INTERFACE IReadOnlyAnalogAnalogInput EXTENDS TOF_Automation.IInputLeafAutomationComponent, TOF_Core.IIOBindable

{attribute 'monitoring' := 'call'}
PROPERTY Converter : IAnalogValueConverter
GET
END_GET
END_PROPERTY

{attribute 'monitoring' := 'call'}
PROPERTY RawValue : LREAL
GET
END_GET
END_PROPERTY

{attribute 'monitoring' := 'call'}
PROPERTY FINAL RawValueType : RAW_ANALOG_VALUE_TYPE
GET
END_GET
END_PROPERTY

{attribute 'monitoring' := 'call'}
PROPERTY Status : REFERENCE TO ANALOG_INPUT_STATUS
GET
END_GET
END_PROPERTY

{attribute 'monitoring' := 'call'}
PROPERTY Value : LREAL
GET
END_GET
END_PROPERTY

END_INTERFACE

(* stored: Version 1.1.0.1
   Itf IReadOnlyAnalogAnalogInput: Id {f18291d7-6e1e-47c5-9cfe-5eb8b3628862}
   Property Converter: Id {38183ee6-a347-4153-bc4c-2d175e7d5e33}
   Get Get: Id {c478d920-13fd-4460-a2cf-cbfd5ab3737e}
   Property RawValue: Id {2bd00137-a6b7-415b-b0ba-8a85a4508031}
   Get Get: Id {1af08222-037d-4c17-824c-b9a38217fe34}
   Property RawValueType: Id {4166ac68-ff2a-4ec2-9aeb-0bae22f15d2f}
   Get Get: Id {4915a80a-e0af-464c-87c8-5de65902eb37}
   Property Status: Id {a079a206-32c1-46c3-a4fe-a37118698c92}
   Get Get: Id {44231e04-1aad-4290-a29c-f0ae5a1c8531}
   Property Value: Id {ee2adc25-672b-4484-9a9d-285dcfba636a}
   Get Get: Id {fbdbf63e-7834-4682-9b6f-7b4bc792058d} *)
